// TIA Portal project "Smart_car_washing_system" (V17)

(* hardware
DEVICE "S7-1500/ET200MP station_1"  S7-1500 station
   slot 0: "Rail_0"  Rack  6ES7 590-1***0-0AA0
   slot 1: "PLC_1"  CPU 1511-1 PN  6ES7 511-1AK00-0AB0  V1.8
      slot 3: "CPU display_1"  6ES7591-1AA00-0AA0
      slot 32768: "PROFINET interface_1"  X1
         slot 32769: "Port_1"  X1 P1
         slot 32770: "Port_2"  X1 P2
*)

// ===== PLC "PLC_1"  CPU 1511-1 PN =====

VAR_GLOBAL   // PLC tag table "Tag table_1"
   "Car_Position_Sensor" AT %I0.0 : Bool;
   "Payment_Authorized" AT %I0.1 : Bool;
   "Emergency_Stop" AT %I0.2 : Bool;
   "Water_Pump" AT %Q0.0 : Bool;
   "Soap_Pump" AT %Q0.1 : Bool;
   "Brush_Motor" AT %Q0.2 : Bool;
   "Rinse_Pump" AT %Q0.3 : Bool;
   "Air_Dryer" AT %Q0.4 : Bool;
   "Completion_Buzzer" AT %Q0.5 : Bool;
   "Water_State" AT %M0.0 : Bool;
   "Soap_Brush_State" AT %M0.1 : Bool;
   "Rinse_State" AT %M0.2 : Bool;
   "Dry_State" AT %M0.3 : Bool;
   "Complete_State" AT %M0.4 : Bool;
END_VAR

// folder: System blocks/Program resources

DATA_BLOCK "Water_Timer"   // DB1
{ S7_Optimized_Access := 'TRUE' }
AUTHOR : Simatic
FAMILY : IEC
NAME : IEC_TMR
VERSION : 1.0
// stored: InstanceOfName IEC_TIMER
"IEC_TIMER"
BEGIN
END_DATA_BLOCK

DATA_BLOCK "Soap_Brush_Timer"   // DB2
{ S7_Optimized_Access := 'TRUE' }
AUTHOR : Simatic
FAMILY : IEC
NAME : IEC_TMR
VERSION : 1.0
// stored: InstanceOfName IEC_TIMER
"IEC_TIMER"
BEGIN
END_DATA_BLOCK

DATA_BLOCK "Rinse_Timer"   // DB3
{ S7_Optimized_Access := 'TRUE' }
AUTHOR : Simatic
FAMILY : IEC
NAME : IEC_TMR
VERSION : 1.0
// stored: InstanceOfName IEC_TIMER
"IEC_TIMER"
BEGIN
END_DATA_BLOCK

DATA_BLOCK "dryer timer"   // DB4
{ S7_Optimized_Access := 'TRUE' }
AUTHOR : Simatic
FAMILY : IEC
NAME : IEC_TMR
VERSION : 1.0
// stored: InstanceOfName IEC_TIMER
"IEC_TIMER"
BEGIN
END_DATA_BLOCK

DATA_BLOCK "Buzzer Timer"   // DB5
{ S7_Optimized_Access := 'TRUE' }
AUTHOR : Simatic
FAMILY : IEC
NAME : IEC_TMR
VERSION : 1.0
// stored: InstanceOfName IEC_TIMER
"IEC_TIMER"
BEGIN
END_DATA_BLOCK

// folder: (top level)

ORGANIZATION_BLOCK "Main"   // OB1, LAD, ProgramCycle
TITLE = "Main Program Sweep (Cycle)"
{ S7_Optimized_Access := 'TRUE' }
VERSION : 0.1
   VAR_INPUT
      Initial_Call : Bool;   // Initial call of this OB
      Remanence : Bool;   // =True, if remanent data are available
   END_VAR
BEGIN

REGION Network 1
   // Start Wash Cycle
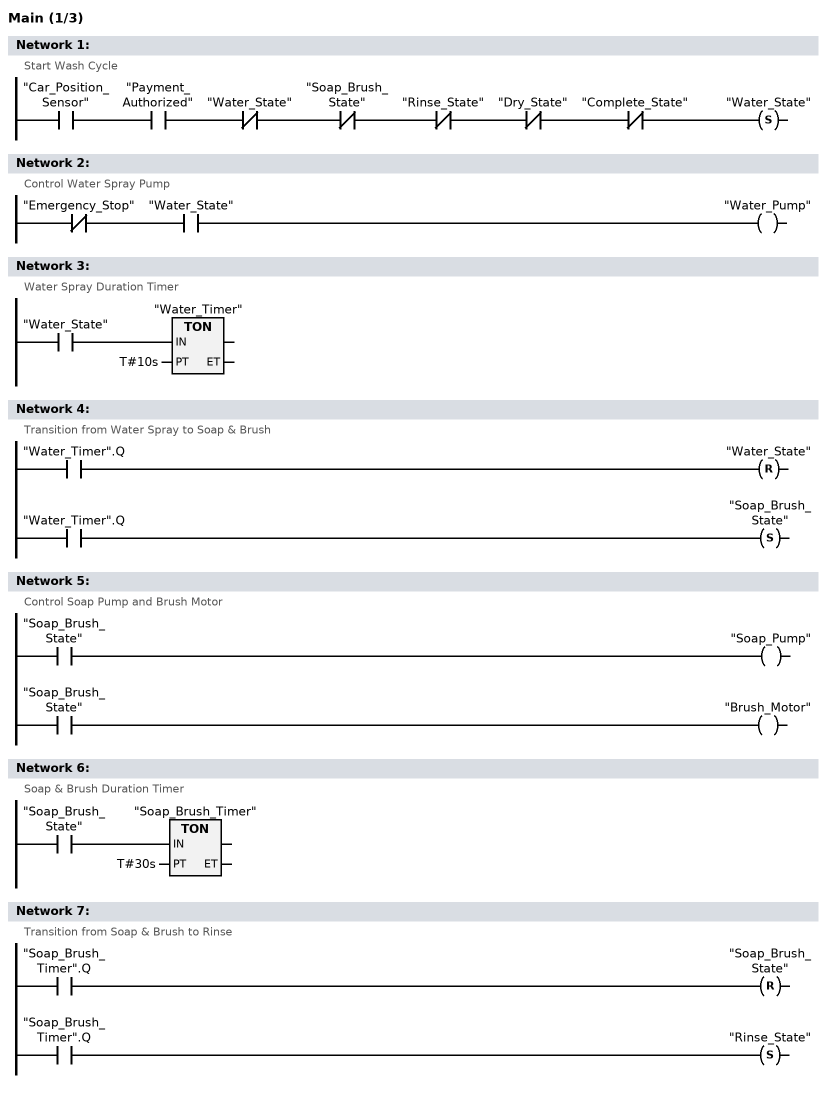
   RUNG wire#powerrail
      Contact( "Car_Position_Sensor" )
      Contact( "Payment_Authorized" )
      I_Contact( "Water_State" )
      I_Contact( "Soap_Brush_State" )
      I_Contact( "Rinse_State" )
      I_Contact( "Dry_State" )
      I_Contact( "Complete_State" )
      S_Coil( "Water_State" )
   END_RUNG
   // the same network as SCL:
   IF "Car_Position_Sensor" AND "Payment_Authorized" AND NOT "Water_State" AND NOT "Soap_Brush_State" AND NOT "Rinse_State" AND NOT "Dry_State" AND NOT "Complete_State" THEN
       "Water_State" := TRUE;
   END_IF;
END_REGION

REGION Network 2
   // Control Water Spray Pump
   RUNG wire#powerrail
      I_Contact( "Emergency_Stop" )
      Contact( "Water_State" )
      Coil( "Water_Pump" )
   END_RUNG
   // the same network as SCL:
   "Water_Pump" := NOT "Emergency_Stop" AND "Water_State";
END_REGION

REGION Network 3
   // Water Spray Duration Timer
   "Water_Timer".TON(IN := "Water_State", PT := T#10s);
END_REGION

REGION Network 4
   // Transition from Water Spray to Soap & Brush
   RUNG wire#powerrail
      Contact( "Water_Timer".Q )
      R_Coil( "Water_State" )
   END_RUNG
   RUNG wire#powerrail
      Contact( "Water_Timer".Q )
      S_Coil( "Soap_Brush_State" )
   END_RUNG
   // the same network as SCL:
   IF "Water_Timer".Q THEN
       "Water_State" := FALSE;
       "Soap_Brush_State" := TRUE;
   END_IF;
END_REGION

REGION Network 5
   // Control Soap Pump and Brush Motor
   RUNG wire#powerrail
      Contact( "Soap_Brush_State" )
      Coil( "Soap_Pump" )
   END_RUNG
   RUNG wire#powerrail
      Contact( "Soap_Brush_State" )
      Coil( "Brush_Motor" )
   END_RUNG
   // the same network as SCL:
   "Soap_Pump" := "Soap_Brush_State";
   "Brush_Motor" := "Soap_Brush_State";
END_REGION

REGION Network 6
   // Soap & Brush Duration Timer
   "Soap_Brush_Timer".TON(IN := "Soap_Brush_State", PT := T#30s);
END_REGION

REGION Network 7
   // Transition from Soap & Brush to Rinse
   RUNG wire#powerrail
      Contact( "Soap_Brush_Timer".Q )
      R_Coil( "Soap_Brush_State" )
   END_RUNG
   RUNG wire#powerrail
      Contact( "Soap_Brush_Timer".Q )
      S_Coil( "Rinse_State" )
   END_RUNG
   // the same network as SCL:
   IF "Soap_Brush_Timer".Q THEN
       "Soap_Brush_State" := FALSE;
       "Rinse_State" := TRUE;
   END_IF;
END_REGION

REGION Network 8
   // Control Rinse Water Pump
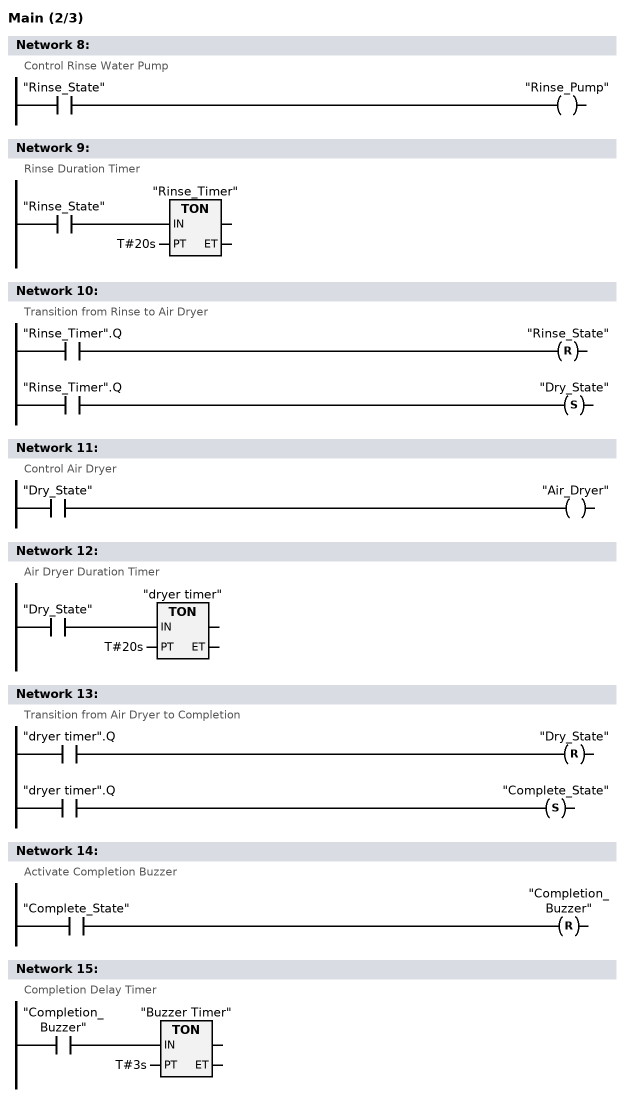
   RUNG wire#powerrail
      Contact( "Rinse_State" )
      Coil( "Rinse_Pump" )
   END_RUNG
   // the same network as SCL:
   "Rinse_Pump" := "Rinse_State";
END_REGION

REGION Network 9
   // Rinse Duration Timer
   "Rinse_Timer".TON(IN := "Rinse_State", PT := T#20s);
END_REGION

REGION Network 10
   // Transition from Rinse to Air Dryer
   RUNG wire#powerrail
      Contact( "Rinse_Timer".Q )
      R_Coil( "Rinse_State" )
   END_RUNG
   RUNG wire#powerrail
      Contact( "Rinse_Timer".Q )
      S_Coil( "Dry_State" )
   END_RUNG
   // the same network as SCL:
   IF "Rinse_Timer".Q THEN
       "Rinse_State" := FALSE;
       "Dry_State" := TRUE;
   END_IF;
END_REGION

REGION Network 11
   // Control Air Dryer
   RUNG wire#powerrail
      Contact( "Dry_State" )
      Coil( "Air_Dryer" )
   END_RUNG
   // the same network as SCL:
   "Air_Dryer" := "Dry_State";
END_REGION

REGION Network 12
   // Air Dryer Duration Timer
   "dryer timer".TON(IN := "Dry_State", PT := T#20s);
END_REGION

REGION Network 13
   // Transition from Air Dryer to Completion
   RUNG wire#powerrail
      Contact( "dryer timer".Q )
      R_Coil( "Dry_State" )
   END_RUNG
   RUNG wire#powerrail
      Contact( "dryer timer".Q )
      S_Coil( "Complete_State" )
   END_RUNG
   // the same network as SCL:
   IF "dryer timer".Q THEN
       "Dry_State" := FALSE;
       "Complete_State" := TRUE;
   END_IF;
END_REGION

REGION Network 14
   // Activate Completion Buzzer
   RUNG wire#powerrail
      Contact( "Complete_State" )
      R_Coil( "Completion_Buzzer" )
   END_RUNG
   // the same network as SCL:
   IF "Complete_State" THEN "Completion_Buzzer" := FALSE; END_IF;
END_REGION

REGION Network 15
   // Completion Delay Timer
   "Buzzer Timer".TON(IN := "Completion_Buzzer", PT := T#3s);
END_REGION

REGION Network 16
   // Reset machine to Idle state
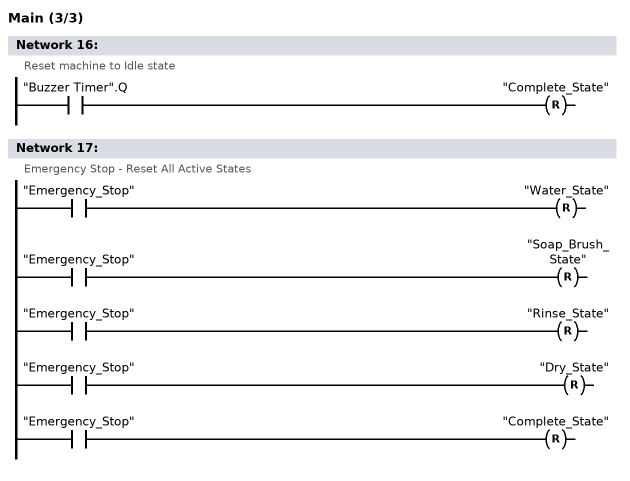
   RUNG wire#powerrail
      Contact( "Buzzer Timer".Q )
      R_Coil( "Complete_State" )
   END_RUNG
   // the same network as SCL:
   IF "Buzzer Timer".Q THEN "Complete_State" := FALSE; END_IF;
END_REGION

REGION Network 17
   // Emergency Stop - Reset All Active States
   RUNG wire#powerrail
      Contact( "Emergency_Stop" )
      R_Coil( "Water_State" )
   END_RUNG
   RUNG wire#powerrail
      Contact( "Emergency_Stop" )
      R_Coil( "Soap_Brush_State" )
   END_RUNG
   RUNG wire#powerrail
      Contact( "Emergency_Stop" )
      R_Coil( "Rinse_State" )
   END_RUNG
   RUNG wire#powerrail
      Contact( "Emergency_Stop" )
      R_Coil( "Dry_State" )
   END_RUNG
   RUNG wire#powerrail
      Contact( "Emergency_Stop" )
      R_Coil( "Complete_State" )
   END_RUNG
   // the same network as SCL:
   IF "Emergency_Stop" THEN
       "Water_State" := FALSE;
       "Soap_Brush_State" := FALSE;
       "Rinse_State" := FALSE;
       "Dry_State" := FALSE;
       "Complete_State" := FALSE;
   END_IF;
END_REGION
END_ORGANIZATION_BLOCK